TYPE HMI_WRN_TemplateMachinePart :
STRUCT
	(*
		Rules:
		Warnings shall only be of type BOOL
		Warnings can be set / reset / activated as you need it (unlike errors!). 
		
		Syntax convention:
		a clear variable name which describes the warning		as described below
		StepLockActive:BOOL;									//Warning [machinepart]: in step modus (steps are held until confirmation the continue to the next step)
	*)
	
	NotRdyRcv_Discharge:BOOL;								//Warning [machinepart]: not ready to receive products
	CameraNotReady:BOOL;									//Warning [machinepart]: waiting for camera ready
END_STRUCT
END_TYPE

(* stored: Version 1.1.0.1
   DUT HMI_WRN_TemplateMachinePart: Id {bc803d7b-969c-46c0-ba3b-c4e157108132} *)
